(* PLC project  *)

CONFIGURATION XI211116
END_CONFIGURATION
